FUNCTION_BLOCK CM_AI_CALL
VAR_INPUT
END_VAR
VAR_OUTPUT
END_VAR
VAR
END_VAR

// NETWORK 1

END_FUNCTION_BLOCK

(* stored: Version 1.1.0.1, ProductVersion 3.1.4024.13
   POU CM_AI_CALL: Id {a0fd4c66-379a-401f-a058-befec02a0903}, SpecialFunc None *)
